// Mitsubishi GX Works2 project: 타이머3   PLC: Q02/Q02H

PROGRAM MAIN
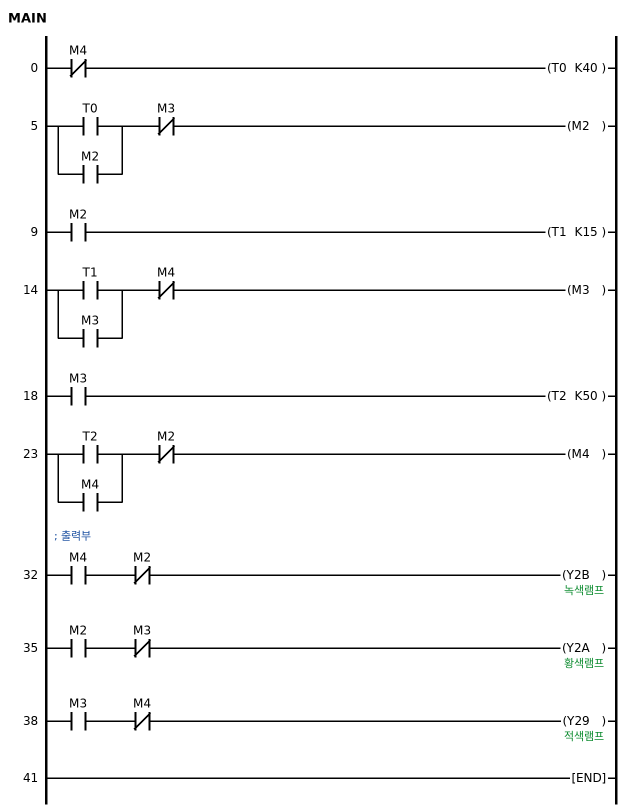
0     LDI     M4
      OUT     T0 K40
5     LD      T0
      OR      M2
      ANI     M3
      OUT     M2
9     LD      M2
      OUT     T1 K15
14    LD      T1
      OR      M3
      ANI     M4
      OUT     M3
18    LD      M3
      OUT     T2 K50
23    LD      T2
      OR      M4
      ANI     M2
      OUT     M4
; 출력부
32    LD      M4
      ANI     M2
      OUT     Y2B  ; 녹색램프
35    LD      M2
      ANI     M3
      OUT     Y2A  ; 황색램프
38    LD      M3
      ANI     M4
      OUT     Y29  ; 적색램프
41    END
END_PROGRAM

// device comments not shown above
X0  ; 공급후진센서
X1  ; 공급전진센서
X2  ; 드릴하강센서
X3  ; 드릴상승센서
X4  ; 송출후진센서
X5  ; 송출전진센서
X0B  ; PB1
X0C  ; PB2
X0D  ; PB3
Y20  ; 공급전진
Y21  ; 공급후진
Y22  ; 드릴하강
Y23  ; 송출전진
Y24  ; 송출후진
Y27  ; 컨베이어
Y28  ; 드릴모터
